TYPE MAIN_BUSY :
(
	eMainWaitStart := 0
);
END_TYPE

(* stored: Version 1.1.0.1, ProductVersion 3.1.4024.2
   DUT MAIN_BUSY: Id {d21a32da-cdbd-493a-ad34-390b23201a84} *)
